//
// This FB reads preasure using up to two PKR 250 sensors, 
// i.e. two instances of FB_CRYO_SENSOR_PKR250.
// The resulting value is a combination of values from available/valid sensors.
// Provides status of each sensor.
// For more info, see method M_SetStatus().
//
FUNCTION_BLOCK FB_CRYO_PRESSURE
VAR_INPUT
	// IMPORTANT NOTE:
	// 		It is assumed that both pressure sensors are of same type.
	//		So, all configuration parameters are same for both sensors.
	//
	{attribute 'OPC.UA.DA' := '0'}
	// Scale factors for each sensor bits -> Volt, U = raw / scale. 
	// Default for 16-bit, +-10V or 0..10V AI: 2^16/10/2 = 3276.8 bit
	in_lrBitsPerVolt_1:	LREAL := 3276.8;	// Scale factor, U = raw / scale. Default 3276.8
	{attribute 'OPC.UA.DA' := '0'}
	in_lrBitsPerVolt_2:	LREAL := 3276.8;	// Scale factor, U = raw / scale. Default 3276.8

	{attribute 'OPC.UA.DA' := '0'}
	in_nType_1:	E_CRYO_SENSOR_TYPE_PRESS	:= E_CRYO_SENSOR_TYPE_PRESS.PKR_250;
	{attribute 'OPC.UA.DA' := '0'}
	in_nType_2:	E_CRYO_SENSOR_TYPE_PRESS	:= E_CRYO_SENSOR_TYPE_PRESS.PKR_250;
	
	
	{attribute 'OPC.UA.DA' := '0'}
	in_lrLimitInVac:	LREAL := 100.0;		// Below this value, the pressure is vacuum
	{attribute 'OPC.UA.DA' := '0'}
	in_lrLimitGoodVac:	LREAL := 10.0E-4;	// Below this value, vacuum is good
	
END_VAR
VAR
	{attribute 'OPC.UA.DA' := '1'}
	Pressure1:	FB_CRYO_SENSOR_PRESSURE;
	{attribute 'OPC.UA.DA' := '1'}
	Pressure2:	FB_CRYO_SENSOR_PRESSURE;
	
	stat:		T_CRYO_PRESSURE_STATUS;	// Complete status
END_VAR

// Get status of two vacuum gauges
M_ReadSensors();

// Set the calculated vacuum pressure
M_SetStatus();

// Get status for both vacuum gauges
METHOD M_ReadSensors
VAR_INPUT
END_VAR
Pressure1(	
	in_nType			:= in_nType_1,
	in_lrBitsPerVolt	:= in_lrBitsPerVolt_1);

Pressure2(	
	in_nType			:= in_nType_2,
	in_lrBitsPerVolt	:= in_lrBitsPerVolt_2);
END_METHOD

// Calculate pressure based on the status of the two sensors
METHOD M_SetStatus
VAR_INPUT
END_VAR
VAR
	lrTmp:		LREAL;	// Temporary var
END_VAR
//
// Determine validity and calculate pressure in user units, i.e. mbar
//
IF Pressure1.stat.bValid  AND  Pressure2.stat.bValid  THEN
	// If any of the two readings are in range, the reading is in range.
	stat.bInRange	:= (Pressure1.stat.bValueInRange  OR  Pressure2.stat.bValueInRange);
	stat.bValid			:= TRUE;
	stat.bWarningSens1	:= FALSE;
	stat.bWarningSens2	:= FALSE;
	
	// Are the readings within 10% from each other
	IF Pressure2.stat.lrPressure > 0.0 THEN
		lrTmp	:= Pressure1.stat.lrPressure / Pressure2.stat.lrPressure;
	ELSE
		lrTmp	:= 0.0;	// Dummy, just to take the higher pressure.
	END_IF
	IF lrTmp > 0.9 AND lrTmp < 1.1  THEN
		// Get the average of the two
		stat.lrPressure	:= (Pressure1.stat.lrPressure + Pressure2.stat.lrPressure) / 2;
	ELSE
		// Get the higher value
		stat.lrPressure	:= MAX(Pressure1.stat.lrPressure, Pressure2.stat.lrPressure);
	END_IF
ELSIF Pressure1.stat.bValid  AND  NOT Pressure2.stat.bValid  THEN
	// Reading of one sensor is OK.
	// However, we set a warning.
	stat.bInRange		:= Pressure1.stat.bValueInRange;
	stat.bValid			:= TRUE;
	stat.bWarningSens1	:= FALSE;
	stat.bWarningSens2	:= TRUE;
	// Take the reading of the first sensor
	stat.lrPressure		:= Pressure1.stat.lrPressure;
ELSIF NOT Pressure1.stat.bValid  AND  Pressure2.stat.bValid  THEN
	// Reading of one sensor is OK.
	// However, we set a warning.
	stat.bInRange		:= Pressure2.stat.bValueInRange;
	stat.bValid			:= TRUE;
	stat.bWarningSens1	:= TRUE;
	stat.bWarningSens2	:= FALSE;
	// Take the reading of the second sensor
	stat.lrPressure		:= Pressure2.stat.lrPressure;
ELSE
	// Both readings are not valid.
	// Reading is not valid.
	stat.bInRange		:= FALSE;
	stat.bValid			:= FALSE;
	stat.bWarningSens1	:= TRUE;
	stat.bWarningSens2	:= TRUE;
	stat.lrPressure		:= 0.0;	// Dummy if reading not valid
END_IF


//
// Set vacuum state based on the pressure level
//
IF NOT stat.bValid  THEN
	stat.bInVacuum		:= FALSE;
	stat.bVacuumGood	:= FALSE;
ELSE
	// 	Check the vacuum levels
	IF stat.lrPressure < in_lrLimitGoodVac  THEN
		stat.bInVacuum		:= TRUE;
		stat.bVacuumGood	:= TRUE;
	ELSIF stat.lrPressure < in_lrLimitInVac  THEN
		stat.bInVacuum		:= TRUE;
		stat.bVacuumGood	:= FALSE;
	ELSE
		stat.bInVacuum		:= FALSE;
		stat.bVacuumGood	:= FALSE;
	END_IF
END_IF
END_METHOD

END_FUNCTION_BLOCK

(* stored: Version 1.1.0.1, ProductVersion 3.1.4024.3
   POU FB_CRYO_PRESSURE: Id {f5f32c8b-8657-4290-adc2-cab6de1506d0}, SpecialFunc None
   Method M_ReadSensors: Id {aec344eb-ec88-4eb3-a458-b87c0e79087d}
   Method M_SetStatus: Id {49dfa7bc-6d77-45c8-b326-ddad265b3d51} *)
